// TIA Portal project "Task 5" (V16)
// Vorlageprojekt für das Buch mit Zielsystem S7-1200

(* hardware
DEVICE "S7-1200-Station_1"  S7-1200 Station
   slot 0: "Baugruppenträger_0"  Rack  V1.0
   slot 1: "PLC_1"  CPU 1211C DC/DC/DC  6ES7 211-1AE40-0XB0  V4.1
*)

// ===== PLC "PLC_1"  CPU 1211C DC/DC/DC =====

VAR_GLOBAL   // PLC tag table "Standard-Variablentabelle"
   "Conv Entry" AT %A0.0 : Bool;
   "Start" AT %E0.0 : Bool;
   "Stop" AT %E0.1 : Bool;
   "X" AT %M0.0 : Bool;
   "Conv Left" AT %Q0.4 : Bool;
   "Conv Right" AT %Q0.5 : Bool;
   "Y(1)" AT %M1.0 : Bool;
   "Load" AT %Q0.1 : Bool;
   "Low Sensor" AT %I0.2 : Bool;
   "Transf Left" AT %Q0.2 : Bool;
   "High Sensor" AT %I0.3 : Bool;
   "Tag_1" AT %M0.1 : Bool;
   "Tag_2" AT %M0.2 : Bool;
   "Left Sensor" AT %I0.5 : Bool;
   "Right Sensor" AT %I0.6 : Bool;
   "Tag_3" AT %M0.3 : Bool;
   "Tag_4" AT %M0.4 : Bool;
   "Transf Right" AT %Q0.3 : Bool;
   "Z" AT %M1.0 : Bool;
   "Tag_5" AT %M1.1 : Bool;
   "Pallet Sensor" AT %I0.7 : Bool;
   "F" AT %M1.4 : Bool;
   "Tag_6" AT %M2.0 : Bool;
   "Tag_7" AT %M2.1 : Bool;
   "A" AT %M3.0 : Bool;
   "B" AT %M3.1 : Bool;
   "T" AT %M3.3 : Bool;
   "R" AT %M3.4 : Bool;
   "Tag_8" AT %M3.6 : Bool;
   "Tag_9" AT %M3.7 : Bool;
   "Tag_10" AT %M4.0 : Bool;
   "Tag_11" AT %M4.1 : Bool;
   "Tag_12" AT %M4.7 : Bool;
END_VAR

// folder: System blocks/Program resources

DATA_BLOCK "T1"   // DB1
{ S7_Optimized_Access := 'TRUE' }
AUTHOR : Simatic
FAMILY : IEC
NAME : IEC_TMR
VERSION : 1.0
// stored: InstanceOfName IEC_TIMER
"IEC_TIMER"
BEGIN
END_DATA_BLOCK

DATA_BLOCK "T2"   // DB2
{ S7_Optimized_Access := 'TRUE' }
AUTHOR : Simatic
FAMILY : IEC
NAME : IEC_TMR
VERSION : 1.0
// stored: InstanceOfName IEC_TIMER
"IEC_TIMER"
BEGIN
END_DATA_BLOCK

DATA_BLOCK "T3"   // DB3
{ S7_Optimized_Access := 'TRUE' }
AUTHOR : Simatic
FAMILY : IEC
NAME : IEC_TMR
VERSION : 1.0
// stored: InstanceOfName IEC_TIMER
"IEC_TIMER"
BEGIN
END_DATA_BLOCK

DATA_BLOCK "T4"   // DB4
{ S7_Optimized_Access := 'TRUE' }
AUTHOR : Simatic
FAMILY : IEC
NAME : IEC_TMR
VERSION : 1.0
// stored: InstanceOfName IEC_TIMER
"IEC_TIMER"
BEGIN
END_DATA_BLOCK

// folder: (top level)

FUNCTION "MHJ-PLC-Lab-Function-S71200" : Void   // FC9000, SCL
{ S7_Optimized_Access := 'TRUE' }
VERSION : 0.1
   VAR_TEMP
      rdTimeReturn : Int;
      outputTime : DTL;
      SyncVal : Byte;
      forVal : Int;
      forVal_2 : Int;
      Value : Byte;
   END_VAR
   VAR CONSTANT
      CompVal : Byte := 16#34;
      Value_01 : Byte := 16#11;
      Value_01_DW : DWord := 16#A165_D992;
      Value_02_DW : DWord := 16#58BE_4401;
   END_VAR
BEGIN

   #Value:=PEEK(area := 16#82,
        dbNumber := 0,
        byteOffset := 511);
   #Value := #Value + 1;

   POKE(area := 16#82,
        dbNumber := 0,
        byteOffset := 511,
        value := #Value);

   POKE(area:=16#81,
        dbNumber:=0,
        byteOffset:=1016,
        value:=#Value_01_DW);
   POKE(area := 16#81,
        dbNumber := 0,
        byteOffset := 1020,
        value := #Value_02_DW);

   POKE(area := 16#81,
        dbNumber := 0,
        byteOffset := 511,
        value := B#16#00);

   FOR #forVal := 0 TO 120 DO
       FOR #forVal_2:=0 TO 10 DO
           #rdTimeReturn:=RD_SYS_T(#outputTime);
           #rdTimeReturn := WR_SYS_T(#outputTime);
           #rdTimeReturn := RD_SYS_T(#outputTime);
           #rdTimeReturn := WR_SYS_T(#outputTime);
       END_FOR;
       #SyncVal:= PEEK(area := 16#81,
                      dbNumber := 0,
                      byteOffset := 511);
       IF #SyncVal = #CompVal THEN
          GOTO M_1;
       END_IF;
   END_FOR;
   RETURN;

   M_1:
   POKE(area := 16#81,
        dbNumber := 0,
        byteOffset := 511,
        value := B#16#0);
END_FUNCTION

ORGANIZATION_BLOCK "Main"   // OB1, LAD, ProgramCycle
TITLE = "Main Program Sweep (Cycle)"
{ S7_Optimized_Access := 'TRUE' }
VERSION : 0.1
   VAR_INPUT
      Initial_Call : Bool;   // Initial call of this OB
      Remanence : Bool;   // =True, if remanent data are available
   END_VAR
   VAR_TEMP   // added for the SCL form of the ladder/FBD networks
      _w1 : Bool;
   END_VAR
BEGIN

REGION Network 1: Konnektierungsbaustein für PLC-Lab
   // Im Netzwerk 1 wird der Konnektierungsbaustein für PLC-Lab aufgerufen.
   // Dieser Aufruf darf nicht entfernt werden!
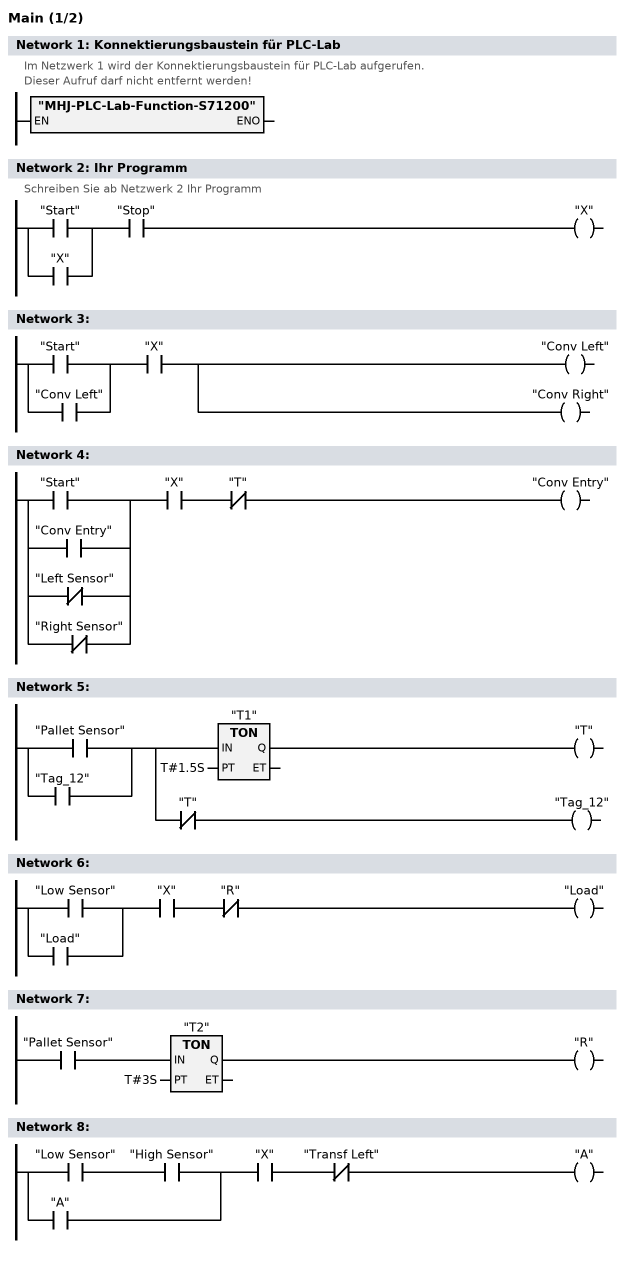
   RUNG wire#powerrail
      "MHJ-PLC-Lab-Function-S71200"()
   END_RUNG
   // the same network as SCL:
   "MHJ-PLC-Lab-Function-S71200"();
END_REGION

REGION Network 2: Ihr Programm
   // Schreiben Sie ab Netzwerk 2 Ihr Programm
   RUNG wire#powerrail
      Contact( "Start" )
      wire#w1
      Contact( "Stop" )
      Coil( "X" )
   END_RUNG
   RUNG wire#powerrail
      Contact( "X" )
   END_RUNG wire#w1
   // the same network as SCL:
   "X" := ("Start" OR "X") AND "Stop";
END_REGION

REGION Network 3
   RUNG wire#powerrail
      Contact( "Start" )
      wire#w1
      Contact( "X" )
      wire#w2
      Coil( "Conv Left" )
   END_RUNG
   RUNG wire#powerrail
      Contact( "Conv Left" )
   END_RUNG wire#w1
   RUNG wire#w2
      Coil( "Conv Right" )
   END_RUNG
   // the same network as SCL:
   "Conv Left" := ("Start" OR "Conv Left") AND "X";
   "Conv Right" := "Conv Left";
END_REGION

REGION Network 4
   RUNG wire#powerrail
      Contact( "Start" )
      wire#w1
      Contact( "X" )
      I_Contact( "T" )
      Coil( "Conv Entry" )
   END_RUNG
   RUNG wire#powerrail
      Contact( "Conv Entry" )
   END_RUNG wire#w1
   RUNG wire#powerrail
      I_Contact( "Left Sensor" )
   END_RUNG wire#w1
   RUNG wire#powerrail
      I_Contact( "Right Sensor" )
   END_RUNG wire#w1
   // the same network as SCL:
   "Conv Entry" := ("Start" OR "Conv Entry" OR NOT "Left Sensor" OR NOT "Right Sensor") AND "X" AND NOT "T";
END_REGION

REGION Network 5
   #_w1 := "Pallet Sensor" OR "Tag_12";
   "T1".TON(IN := #_w1, PT := T#1.5S);
   "T" := "T1".Q;
   "Tag_12" := #_w1 AND NOT "T";
END_REGION

REGION Network 6
   RUNG wire#powerrail
      Contact( "Low Sensor" )
      wire#w1
      Contact( "X" )
      I_Contact( "R" )
      Coil( "Load" )
   END_RUNG
   RUNG wire#powerrail
      Contact( "Load" )
   END_RUNG wire#w1
   // the same network as SCL:
   "Load" := ("Low Sensor" OR "Load") AND "X" AND NOT "R";
END_REGION

REGION Network 7
   "T2".TON(IN := "Pallet Sensor", PT := T#3S);
   "R" := "T2".Q;
END_REGION

REGION Network 8
   RUNG wire#powerrail
      Contact( "Low Sensor" )
      Contact( "High Sensor" )
      wire#w1
      Contact( "X" )
      I_Contact( "Transf Left" )
      Coil( "A" )
   END_RUNG
   RUNG wire#powerrail
      Contact( "A" )
   END_RUNG wire#w1
   // the same network as SCL:
   "A" := (("Low Sensor" AND "High Sensor") OR "A") AND "X" AND NOT "Transf Left";
END_REGION

REGION Network 9
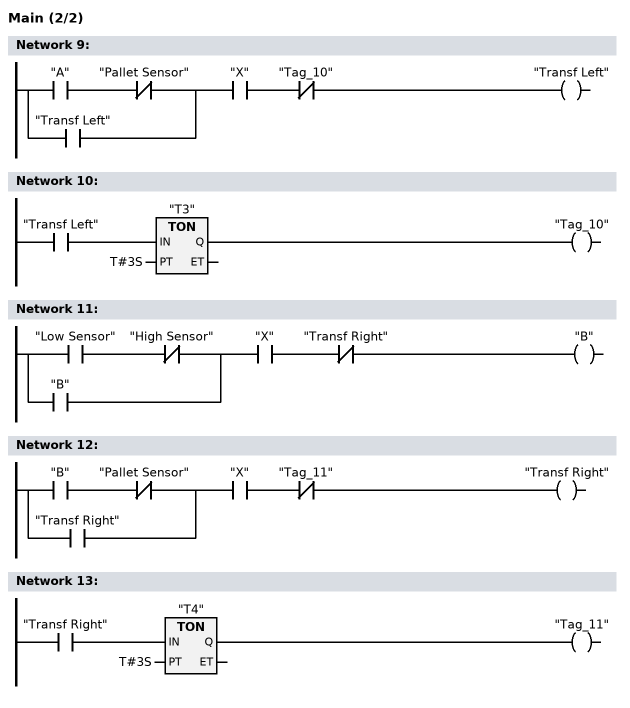
   RUNG wire#powerrail
      Contact( "A" )
      I_Contact( "Pallet Sensor" )
      wire#w1
      Contact( "X" )
      I_Contact( "Tag_10" )
      Coil( "Transf Left" )
   END_RUNG
   RUNG wire#powerrail
      Contact( "Transf Left" )
   END_RUNG wire#w1
   // the same network as SCL:
   "Transf Left" := (("A" AND NOT "Pallet Sensor") OR "Transf Left") AND "X" AND NOT "Tag_10";
END_REGION

REGION Network 10
   "T3".TON(IN := "Transf Left", PT := T#3S);
   "Tag_10" := "T3".Q;
END_REGION

REGION Network 11
   RUNG wire#powerrail
      Contact( "Low Sensor" )
      I_Contact( "High Sensor" )
      wire#w1
      Contact( "X" )
      I_Contact( "Transf Right" )
      Coil( "B" )
   END_RUNG
   RUNG wire#powerrail
      Contact( "B" )
   END_RUNG wire#w1
   // the same network as SCL:
   "B" := (("Low Sensor" AND NOT "High Sensor") OR "B") AND "X" AND NOT "Transf Right";
END_REGION

REGION Network 12
   RUNG wire#powerrail
      Contact( "B" )
      I_Contact( "Pallet Sensor" )
      wire#w1
      Contact( "X" )
      I_Contact( "Tag_11" )
      Coil( "Transf Right" )
   END_RUNG
   RUNG wire#powerrail
      Contact( "Transf Right" )
   END_RUNG wire#w1
   // the same network as SCL:
   "Transf Right" := (("B" AND NOT "Pallet Sensor") OR "Transf Right") AND "X" AND NOT "Tag_11";
END_REGION

REGION Network 13
   "T4".TON(IN := "Transf Right", PT := T#3S);
   "Tag_11" := "T4".Q;
END_REGION
END_ORGANIZATION_BLOCK